(* IEC 61131-3 sources: PLC-Programming-with-Ladder-Logic-Mini-Project/Solutions/openplc/part4b, 1 file *)

(* ---- part4b.st ---- *)
PROGRAM CarParkingControl
    VAR
        Main_Switch : BOOL;
        Car_In_Lane : BOOL;
        Green_Light : BOOL;
        Red_Light : BOOL;
        Car_Counter : INT;
    END_VAR

    IF Main_Switch THEN
        IF Car_Counter >= 4 THEN
            Red_Light := TRUE;
            Green_Light := FALSE;
        ELSIF Car_In_Lane THEN
            Red_Light := TRUE;
            Green_Light := FALSE;
            Car_Counter := Car_Counter + 1;
        ELSE
            Green_Light := TRUE;
            Red_Light := FALSE;
            IF Car_Counter > 0 THEN
                Car_Counter := Car_Counter - 1;
            END_IF;
        END_IF;
    ELSE
        Red_Light := FALSE;
        Green_Light := FALSE;
    END_IF;
END_PROGRAM

CONFIGURATION Config0
    RESOURCE Res0 ON PLC
        TASK task0(INTERVAL := T#20ms, PRIORITY := 0);
        PROGRAM instance0 WITH task0 : CarParkingControl;
    END_RESOURCE
END_CONFIGURATION
